PROGRAM POU
VAR
END_VAR

END_PROGRAM

(* stored: Version 1.1.0.1, ProductVersion 3.1.4024.13
   POU POU: Id {985b0e46-eb1a-4116-9796-15cdb41b0793}, SpecialFunc None *)
